(* IEC 61131-3 sources: repolevel_ST_code_completion/output/full_case_fixed/repoeval_VisuElements/readful_result_history, 11 files *)

(* ---- RotationCalculation_0.st ---- *)
FUNCTION RotationCalculation : BOOL
VAR_INPUT
    rCenterX : REAL;    (* X coordinate of rotation center *)
    rCenterY : REAL;    (* Y coordinate of rotation center *)
    rAngle : REAL;      (* Rotation angle in degrees *)
    rPointX : REAL;     (* X coordinate of point to rotate *)
    rPointY : REAL;     (* Y coordinate of point to rotate *)
END_VAR

VAR_OUTPUT
    rRotatedX : REAL;   (* X coordinate after rotation *)
    rRotatedY : REAL;   (* Y coordinate after rotation *)
END_VAR
VAR
    rRadians : REAL;
    rCos : REAL;
    rSin : REAL;
    rTranslatedX : REAL;
    rTranslatedY : REAL;
END_VAR

rRadians := rAngle * PI / 180; (* Convert angle to radians *)
rCos := COS(rRadians);         (* Calculate cosine of the angle *)
rSin := SIN(rRadians);         (* Calculate sine of the angle *)

(* Translate point to origin relative to the center *)
rTranslatedX := rPointX - rCenterX;
rTranslatedY := rPointY - rCenterY;

(* Rotate the point *)
rRotatedX := rTranslatedX * rCos - rTranslatedY * rSin + rCenterX;
rRotatedY := rTranslatedX * rSin + rTranslatedY * rCos + rCenterY;

RETURN TRUE; (* Indicate successful calculation *)
END_FUNCTION

(* ---- RotationCalculation_1.st ---- *)
FUNCTION RotationCalculation : BOOL
VAR_INPUT
    rCenterX : REAL;    (* X coordinate of rotation center *)
    rCenterY : REAL;    (* Y coordinate of rotation center *)
    rAngle : REAL;      (* Rotation angle in degrees *)
    rPointX : REAL;     (* X coordinate of point to rotate *)
    rPointY : REAL;     (* Y coordinate of point to rotate *)
END_VAR

VAR_OUTPUT
    rRotatedX : REAL;   (* X coordinate after rotation *)
    rRotatedY : REAL;   (* Y coordinate after rotation *)
END_VAR
VAR
    rRadians : REAL;
    rCos : REAL;
    rSin : REAL;
    rTranslatedX : REAL;
    rTranslatedY : REAL;
END_VAR

rRadians := rAngle * PI / 180; (* Convert angle to radians *)
rCos := COS(rRadians);         (* Calculate cosine of the angle *)
rSin := SIN(rRadians);         (* Calculate sine of the angle *)

(* Translate point to origin relative to the center *)
rTranslatedX := rPointX - rCenterX;
rTranslatedY := rPointY - rCenterY;

(* Rotate the point *)
rRotatedX := rTranslatedX * rCos - rTranslatedY * rSin + rCenterX;
rRotatedY := rTranslatedX * rSin + rTranslatedY * rCos + rCenterY;

RotationCalculation := TRUE; // Assigning the result value to the function's name
  RETURN; // Explicit return without a value
END_FUNCTION

(* ---- RotationCalculation_2.st ---- *)
FUNCTION RotationCalculation : BOOL
VAR_INPUT
    rCenterX : REAL;    (* X coordinate of rotation center *)
    rCenterY : REAL;    (* Y coordinate of rotation center *)
    rAngle : REAL;      (* Rotation angle in degrees *)
    rPointX : REAL;     (* X coordinate of point to rotate *)
    rPointY : REAL;     (* Y coordinate of point to rotate *)
END_VAR

VAR_OUTPUT
    rRotatedX : REAL;   (* X coordinate after rotation *)
    rRotatedY : REAL;   (* Y coordinate after rotation *)
END_VAR
VAR
    rRadians : REAL;
    rCos : REAL;
    rSin : REAL;
    rTranslatedX : REAL;
    rTranslatedY : REAL;
END_VAR

rRadians := rAngle * 3.141592653589793 / 180; // Manually replace PI with its approximate value
rCos := COS(rRadians);         (* Calculate cosine of the angle *)
rSin := SIN(rRadians);         (* Calculate sine of the angle *)

(* Translate point to origin relative to the center *)
rTranslatedX := rPointX - rCenterX;
rTranslatedY := rPointY - rCenterY;

(* Rotate the point *)
rRotatedX := rTranslatedX * rCos - rTranslatedY * rSin + rCenterX;
rRotatedY := rTranslatedX * rSin + rTranslatedY * rCos + rCenterY;

RotationCalculation := TRUE; // Assigning the result value to the function's name
  RETURN; // Explicit return without a value
END_FUNCTION

(* ---- MouseEventHandler_0.st ---- *)
FUNCTION_BLOCK MouseEventHandler
VAR_INPUT
    xLeftClick : BOOL;      (* Left mouse button click *)
    xRightClick : BOOL;     (* Right mouse button click *)
    xMiddleClick : BOOL;    (* Middle mouse button click *)
    xMouseMove : BOOL;      (* Mouse movement detected *)
    rMouseX : REAL;         (* Current mouse X position *)
    rMouseY : REAL;         (* Current mouse Y position *)
    tDblClickTime : TIME := T#300MS;  (* Double click timeout *)
END_VAR

VAR_OUTPUT
    eMouseEvent : INT;      (* Event type: 0=None, 1=SingleClick, 2=DoubleClick, 3=RightClick, 4=MiddleClick *)
    rEventX : REAL;         (* X position where event occurred *)
    rEventY : REAL;         (* Y position where event occurred *)
    xEventActive : BOOL;    (* TRUE when an event is active *)
END_VAR
VAR
    LeftClickTimer : TON;
    xLeftClickOld : BOOL;
    iClickCount : INT := 0;
    xEventProcessed : BOOL := FALSE;
END_VAR

(* Reset event state *)
eMouseEvent := 0;
xEventActive := FALSE;

(* Handle left click events (single/double click) *)
IF xLeftClick AND NOT xLeftClickOld THEN
    (* First click detected *)
    IF iClickCount = 0 THEN
        LeftClickTimer(IN := TRUE, PT := tDblClickTime);
        iClickCount := 1;
    ELSE
        (* Second click within time window *)
        LeftClickTimer(IN := FALSE);
        eMouseEvent := 2; (* Double click *)
        rEventX := rMouseX;
        rEventY := rMouseY;
        xEventActive := TRUE;
        iClickCount := 0;
        xEventProcessed := TRUE;
    END_IF
ELSIF NOT xLeftClick AND xLeftClickOld THEN
    (* Left button released *)
    IF iClickCount = 1 AND NOT xEventProcessed THEN
        LeftClickTimer();
        IF NOT LeftClickTimer.Q THEN
            (* Still waiting for potential double click *)
            (* Will be handled by timer logic below *)
        END_IF
    END_IF
END_IF

(* Check for double click timeout *)
IF LeftClickTimer.Q AND iClickCount = 1 THEN
    eMouseEvent := 1; (* Single click *)
    rEventX := rMouseX;
    rEventY := rMouseY;
    xEventActive := TRUE;
    iClickCount := 0;
END_IF

(* Handle right click events *)
IF xRightClick THEN
    eMouseEvent := 3; (* Right click *)
    rEventX := rMouseX;
    rEventY := rMouseY;
    xEventActive := TRUE;
END_IF

(* Handle middle click events *)
IF xMiddleClick THEN
    eMouseEvent := 4; (* Middle click *)
    rEventX := rMouseX;
    rEventY := rMouseY;
    xEventActive := TRUE;
END_IF

(* Handle mouse movement events *)
IF xMouseMove THEN
    eMouseEvent := 0; (* Mouse movement does not trigger an event *)
    rEventX := rMouseX;
    rEventY := rMouseY;
    xEventActive := FALSE;
END_IF

(* Update old state *)
xLeftClickOld := xLeftClick;
END_FUNCTION_BLOCK

(* ---- MouseEventHandler_1.st ---- *)
FUNCTION_BLOCK MouseEventHandler
VAR_INPUT
    xLeftClick : BOOL;      (* Left mouse button click *)
    xRightClick : BOOL;     (* Right mouse button click *)
    xMiddleClick : BOOL;    (* Middle mouse button click *)
    xMouseMove : BOOL;      (* Mouse movement detected *)
    rMouseX : REAL;         (* Current mouse X position *)
    rMouseY : REAL;         (* Current mouse Y position *)
    tDblClickTime : TIME := T#300MS;  (* Double click timeout *)
END_VAR

VAR_OUTPUT
    eMouseEvent : INT;      (* Event type: 0=None, 1=SingleClick, 2=DoubleClick, 3=RightClick, 4=MiddleClick *)
    rEventX : REAL;         (* X position where event occurred *)
    rEventY : REAL;         (* Y position where event occurred *)
    xEventActive : BOOL;    (* TRUE when an event is active *)
END_VAR
VAR
    LeftClickTimer : TON;
    xLeftClickOld : BOOL;
    iClickCount : INT := 0;
    xEventProcessed : BOOL := FALSE;
END_VAR

(* Reset event state *)
eMouseEvent := 0;
xEventActive := FALSE;

(* Handle left click events (single/double click) *)
IF xLeftClick AND NOT xLeftClickOld THEN
    (* First click detected *)
    IF iClickCount = 0 THEN
        LeftClickTimer(IN := TRUE, PT := tDblClickTime);
        iClickCount := 1;
    ELSE
        (* Second click within time window *)
        LeftClickTimer(IN := FALSE);
        eMouseEvent := 2; (* Double click *)
        rEventX := rMouseX;
        rEventY := rMouseY;
        xEventActive := TRUE;
        iClickCount := 0;
        xEventProcessed := TRUE;
    END_IF
ELSIF NOT xLeftClick AND xLeftClickOld THEN
    (* Left button released *)
    IF iClickCount = 1 AND NOT xEventProcessed THEN
LeftClickTimer(IN := FALSE, PT := T#0MS); // Reset the timer properly
        IF NOT LeftClickTimer.Q THEN
            (* Still waiting for potential double click *)
            (* Will be handled by timer logic below *)
        END_IF
    END_IF
END_IF

(* Check for double click timeout *)
IF LeftClickTimer.Q AND iClickCount = 1 THEN
    eMouseEvent := 1; (* Single click *)
    rEventX := rMouseX;
    rEventY := rMouseY;
    xEventActive := TRUE;
    iClickCount := 0;
END_IF

(* Handle right click events *)
IF xRightClick THEN
    eMouseEvent := 3; (* Right click *)
    rEventX := rMouseX;
    rEventY := rMouseY;
    xEventActive := TRUE;
END_IF

(* Handle middle click events *)
IF xMiddleClick THEN
    eMouseEvent := 4; (* Middle click *)
    rEventX := rMouseX;
    rEventY := rMouseY;
    xEventActive := TRUE;
END_IF

(* Handle mouse movement events *)
IF xMouseMove THEN
    eMouseEvent := 0; (* Mouse movement does not trigger an event *)
    rEventX := rMouseX;
    rEventY := rMouseY;
    xEventActive := FALSE;
END_IF

(* Update old state *)
xLeftClickOld := xLeftClick;
END_FUNCTION_BLOCK

(* ---- MouseEventHandler_2.st ---- *)
FUNCTION_BLOCK MouseEventHandler
VAR_INPUT
    xLeftClick : BOOL;      (* Left mouse button click *)
    xRightClick : BOOL;     (* Right mouse button click *)
    xMiddleClick : BOOL;    (* Middle mouse button click *)
    xMouseMove : BOOL;      (* Mouse movement detected *)
    rMouseX : REAL;         (* Current mouse X position *)
    rMouseY : REAL;         (* Current mouse Y position *)
    tDblClickTime : TIME := T#300MS;  (* Double click timeout *)
END_VAR

VAR_OUTPUT
    eMouseEvent : INT;      (* Event type: 0=None, 1=SingleClick, 2=DoubleClick, 3=RightClick, 4=MiddleClick *)
    rEventX : REAL;         (* X position where event occurred *)
    rEventY : REAL;         (* Y position where event occurred *)
    xEventActive : BOOL;    (* TRUE when an event is active *)
END_VAR
VAR
    LeftClickTimer : TON;
    xLeftClickOld : BOOL;
    iClickCount : INT := 0;
    xEventProcessed : BOOL := FALSE;
END_VAR

(* Reset event state *)
eMouseEvent := 0;
xEventActive := FALSE;

(* Handle left click events (single/double click) *)
IF xLeftClick AND NOT xLeftClickOld THEN
    (* First click detected *)
    IF iClickCount = 0 THEN
        LeftClickTimer(IN := TRUE, PT := tDblClickTime);
        iClickCount := 1;
    ELSE
        (* Second click within time window *)
        LeftClickTimer(IN := FALSE);
        eMouseEvent := 2; (* Double click *)
        rEventX := rMouseX;
        rEventY := rMouseY;
        xEventActive := TRUE;
        iClickCount := 0;
        xEventProcessed := TRUE;
    END_IF
ELSIF NOT xLeftClick AND xLeftClickOld THEN
    (* Left button released *)
    IF iClickCount = 1 AND NOT xEventProcessed THEN
LeftClickTimer(IN := FALSE); // Simplified reset; PT remains unchanged
        IF NOT LeftClickTimer.Q THEN
            (* Still waiting for potential double click *)
            (* Will be handled by timer logic below *)
        END_IF
    END_IF
END_IF

(* Check for double click timeout *)
IF LeftClickTimer.Q AND iClickCount = 1 THEN
    eMouseEvent := 1; (* Single click *)
    rEventX := rMouseX;
    rEventY := rMouseY;
    xEventActive := TRUE;
    iClickCount := 0;
END_IF

(* Handle right click events *)
IF xRightClick THEN
    eMouseEvent := 3; (* Right click *)
    rEventX := rMouseX;
    rEventY := rMouseY;
    xEventActive := TRUE;
END_IF

(* Handle middle click events *)
IF xMiddleClick THEN
    eMouseEvent := 4; (* Middle click *)
    rEventX := rMouseX;
    rEventY := rMouseY;
    xEventActive := TRUE;
END_IF

(* Handle mouse movement events *)
IF xMouseMove THEN
    eMouseEvent := 0; (* Mouse movement does not trigger an event *)
    rEventX := rMouseX;
    rEventY := rMouseY;
    xEventActive := FALSE;
END_IF

(* Update old state *)
xLeftClickOld := xLeftClick;
END_FUNCTION_BLOCK

(* ---- MouseEventHandler_3.st ---- *)
FUNCTION_BLOCK MouseEventHandler
VAR_INPUT
    xLeftClick : BOOL;      (* Left mouse button click *)
    xRightClick : BOOL;     (* Right mouse button click *)
    xMiddleClick : BOOL;    (* Middle mouse button click *)
    xMouseMove : BOOL;      (* Mouse movement detected *)
    rMouseX : REAL;         (* Current mouse X position *)
    rMouseY : REAL;         (* Current mouse Y position *)
    tDblClickTime : TIME := T#300MS;  (* Double click timeout *)
END_VAR

VAR_OUTPUT
    eMouseEvent : INT;      (* Event type: 0=None, 1=SingleClick, 2=DoubleClick, 3=RightClick, 4=MiddleClick *)
    rEventX : REAL;         (* X position where event occurred *)
    rEventY : REAL;         (* Y position where event occurred *)
    xEventActive : BOOL;    (* TRUE when an event is active *)
END_VAR
VAR
    LeftClickTimer : TON;
    xLeftClickOld : BOOL;
    iClickCount : INT := 0;
    xEventProcessed : BOOL := FALSE;
END_VAR

(* Reset event state *)
eMouseEvent := 0;
xEventActive := FALSE;

(* Handle left click events (single/double click) *)
IF xLeftClick AND NOT xLeftClickOld THEN
    (* First click detected *)
    IF iClickCount = 0 THEN
        LeftClickTimer(IN := TRUE, PT := tDblClickTime);
        iClickCount := 1;
    ELSE
        (* Second click within time window *)
// Simplify reset logic
    LeftClickTimer(IN := FALSE); // Keep, but ensure timer conditions are respected elsewhere
        eMouseEvent := 2; (* Double click *)
        rEventX := rMouseX;
        rEventY := rMouseY;
        xEventActive := TRUE;
        iClickCount := 0;
        xEventProcessed := TRUE;
    END_IF
ELSIF NOT xLeftClick AND xLeftClickOld THEN
    (* Left button released *)
    IF iClickCount = 1 AND NOT xEventProcessed THEN
LeftClickTimer(IN := FALSE); // Simplified reset; PT remains unchanged
        IF NOT LeftClickTimer.Q THEN
            (* Still waiting for potential double click *)
            (* Will be handled by timer logic below *)
        END_IF
    END_IF
END_IF

(* Check for double click timeout *)
IF LeftClickTimer.Q AND iClickCount = 1 THEN
    eMouseEvent := 1; (* Single click *)
    rEventX := rMouseX;
    rEventY := rMouseY;
    xEventActive := TRUE;
    iClickCount := 0;
END_IF

(* Handle right click events *)
IF xRightClick THEN
    eMouseEvent := 3; (* Right click *)
    rEventX := rMouseX;
    rEventY := rMouseY;
    xEventActive := TRUE;
END_IF

(* Handle middle click events *)
IF xMiddleClick THEN
    eMouseEvent := 4; (* Middle click *)
    rEventX := rMouseX;
    rEventY := rMouseY;
    xEventActive := TRUE;
END_IF

(* Handle mouse movement events *)
IF xMouseMove THEN
    eMouseEvent := 0; (* Mouse movement does not trigger an event *)
    rEventX := rMouseX;
    rEventY := rMouseY;
    xEventActive := FALSE;
END_IF

(* Update old state *)
xLeftClickOld := xLeftClick;
END_FUNCTION_BLOCK

(* ---- NodeExpandCollapse_0.st ---- *)
FUNCTION_BLOCK NodeExpandCollapse
VAR_INPUT
    xNodeClick : BOOL;  (* Input signal for node click *)
    tDblClickTime : TIME := T#500MS;  (* Time to wait for double click *)
END_VAR

VAR_OUTPUT
    xNodeExpand : BOOL;  (* Output: TRUE when node is expanded *)
    xNodeSelected : BOOL; (* Output: TRUE when node is selected *)
END_VAR
VAR
    NodeDblClick : TON;
    xNodeClickOld : BOOL;
    iNodeState : INT := 1;
END_VAR

CASE iNodeState OF
    1: (* Wait for first click *)
        IF xNodeClick AND NOT xNodeClickOld THEN
            NodeDblClick(IN := TRUE, PT := tDblClickTime);
            iNodeState := 2;
            xNodeSelected := TRUE;
        END_IF

    2: (* Wait for second click or timeout *)
        NodeDblClick();
        IF NodeDblClick.Q THEN
            (* Timeout - single click, reset *)
            NodeDblClick(IN := FALSE);
            xNodeClickOld := FALSE;
            iNodeState := 1;
            xNodeSelected := FALSE;
        ELSIF NOT xNodeClick AND xNodeClickOld THEN
            (* Second click detected - toggle expansion *)
            NodeDblClick(IN := FALSE);
            xNodeExpand := NOT xNodeExpand;
            iNodeState := 1;
            xNodeSelected := FALSE;
        END_IF
END_CASE

xNodeClickOld := xNodeClick;
END_FUNCTION_BLOCK

(* ---- NodeExpandCollapse_1.st ---- *)
FUNCTION_BLOCK NodeExpandCollapse
VAR_INPUT
    xNodeClick : BOOL;  (* Input signal for node click *)
    tDblClickTime : TIME := T#500MS;  (* Time to wait for double click *)
END_VAR

VAR_OUTPUT
    xNodeExpand : BOOL;  (* Output: TRUE when node is expanded *)
    xNodeSelected : BOOL; (* Output: TRUE when node is selected *)
END_VAR
VAR
    NodeDblClick : TON;
    xNodeClickOld : BOOL;
    iNodeState : INT := 1;
END_VAR

CASE iNodeState OF
    1: (* Wait for first click *)
        IF xNodeClick AND NOT xNodeClickOld THEN
            NodeDblClick(IN := TRUE, PT := tDblClickTime);
            iNodeState := 2;
            xNodeSelected := TRUE;
        END_IF

    2: (* Wait for second click or timeout *)
NodeDblClick(IN := TRUE, PT := tDblClickTime); // Properly call TON instance with parameters
    IF NodeDblClick.Q THEN
      (* Timeout - single click, reset *)
      NodeDblClick(IN := FALSE, PT := T#0S); // Gracefully reset the TON block
      xNodeClickOld := FALSE;  // Reset click state properly
      iNodeState := 1;          // Reset the state
      xNodeSelected := FALSE;   // Reset selection to inactive
    ELSIF NOT xNodeClick AND xNodeClickOld THEN
      (* Second click detected - toggle expansion *)
      NodeDblClick(IN := FALSE, PT := T#0S); // Gracefully stop TON instance
      xNodeExpand := NOT xNodeExpand;      // Toggle the expansion state
      iNodeState := 1;                     // Reset the state
      xNodeSelected := FALSE;              // Reset selection to inactive
    END_IF
END_CASE

xNodeClickOld := xNodeClick;
END_FUNCTION_BLOCK

(* ---- NodeExpandCollapse_2.st ---- *)
FUNCTION_BLOCK NodeExpandCollapse
VAR_INPUT
    xNodeClick : BOOL;  (* Input signal for node click *)
    tDblClickTime : TIME := T#500MS;  (* Time to wait for double click *)
END_VAR

VAR_OUTPUT
    xNodeExpand : BOOL;  (* Output: TRUE when node is expanded *)
    xNodeSelected : BOOL; (* Output: TRUE when node is selected *)
END_VAR
VAR
    NodeDblClick : TON;
    xNodeClickOld : BOOL;
    iNodeState : INT := 1;
END_VAR

CASE iNodeState OF
    1: (* Wait for first click *)
        IF xNodeClick AND NOT xNodeClickOld THEN
            NodeDblClick(IN := TRUE, PT := tDblClickTime);
            iNodeState := 2;
            xNodeSelected := TRUE;
        END_IF

    2: (* Wait for second click or timeout *)
IF NodeDblClick.Q THEN
 (* Timeout - single click, reset *)
 NodeDblClick(IN := FALSE); // Stop the TON block without modifying PT
 xNodeClickOld := FALSE;    // Reset click state properly
 iNodeState := 1;           // Reset the state
 xNodeSelected := FALSE;    // Reset selection to inactive
ELSIF NOT xNodeClick AND xNodeClickOld THEN
 (* Second click detected - toggle expansion *)
 NodeDblClick(IN := FALSE); // Stop the TON block without modifying PT
 xNodeExpand := NOT xNodeExpand; // Toggle the expansion state
 iNodeState := 1;                // Reset the state
 xNodeSelected := FALSE;         // Reset selection to inactive
END_IF
END_CASE

xNodeClickOld := xNodeClick;
END_FUNCTION_BLOCK

(* ---- NodeExpandCollapse_3.st ---- *)
FUNCTION_BLOCK NodeExpandCollapse
VAR_INPUT
    xNodeClick : BOOL;  (* Input signal for node click *)
    tDblClickTime : TIME := T#500MS;  (* Time to wait for double click *)
END_VAR

VAR_OUTPUT
    xNodeExpand : BOOL;  (* Output: TRUE when node is expanded *)
    xNodeSelected : BOOL; (* Output: TRUE when node is selected *)
END_VAR
VAR
    NodeDblClick : TON;
    xNodeClickOld : BOOL;
    iNodeState : INT := 1;
END_VAR

CASE iNodeState OF
    1: (* Wait for first click *)
        IF xNodeClick AND NOT xNodeClickOld THEN
            NodeDblClick(IN := TRUE, PT := tDblClickTime);
            iNodeState := 2;
            xNodeSelected := TRUE;
        END_IF

    2: (* Wait for second click or timeout *)
NodeDblClick(IN := TRUE, PT := tDblClickTime); // Ensure TON block execution for timing
IF NodeDblClick.Q THEN
(* Timeout - single click, reset *)
NodeDblClick(IN := FALSE); // Stop the TON block without modifying PT
xNodeClickOld := FALSE;    // Reset click state properly
iNodeState := 1;           // Reset the state
xNodeSelected := FALSE;    // Reset selection to inactive
ELSIF NOT xNodeClick AND xNodeClickOld THEN
(* Second click detected - toggle expansion *)
NodeDblClick(IN := FALSE); // Stop the TON block without modifying PT
xNodeExpand := NOT xNodeExpand; // Toggle the expansion state
iNodeState := 1;                // Reset the state
xNodeSelected := FALSE;         // Reset selection to inactive
END_IF
END_CASE

xNodeClickOld := xNodeClick;
END_FUNCTION_BLOCK
